(* IEC 61131-3 sources: POMIRTS_lab3/AS/Library_2/ArEthBond, 3 files *)

(* ---- ArEthBond.typ ---- *)
 TYPE
	ArEthBondStateType : STRUCT											(*status data of a bond*)
		ActiveDevice 						: STRING[128];				(*name of the currently active device*)
		PrimaryLinkStatus 					: UDINT;					(*link status of the primary device*)
		SecondaryLinkStatus 				: UDINT;					(*link status of the secondary device*)
		NumberArpReachedTargets 			: UDINT;					(*number of currently reached ARP targets*)
	END_STRUCT;

	ArEthBondStatisticsType : STRUCT									(*statistical data of a bond*)
		SwitchCount 						: UDINT; 					(*number of occurred switches*)
		PrimaryLinkErrorCount 				: UDINT;					(*number of link errors of the primary device*)
		SecondaryLinkErrorCount 			: UDINT;					(*number of link errors of the secondary device*)
		PrimaryArpErrorCount 				: UDINT;					(*number of ARP errors of the primary device*)
		SecondaryArpErrorCount 				: UDINT;					(*number of ARP errors of the secondary device*)
		LastErrorUtcTimeStampSeconds 		: UDINT;					(*seconds part of the last error time stamp*)
		LastErrorUtcTimeStampNanoSeconds 	: UDINT;					(*nano seconds part of the last error time stamp*)
	END_STRUCT;

	ArEthBondConfigurationType : STRUCT
		ArpMonitorPeriodMs 					: UDINT; 					(*period of the ARP monitoring in ms*)
		NumberArpConfiguredTargets 			: UDINT; 					(*number of configured ARP targets*)
	END_STRUCT;

	ArEthBondInternalType : STRUCT
		FBStateCtx							: ArFBStateInternalType; 	(*internal status*)
	END_STRUCT;
END_TYPE

(* ---- ArEthBond.var ---- *)
 VAR CONSTANT
	arETHBOND_ERR_INVALID_NAME 	: DINT := -1070585906;	(*invalid bond name as input parameter*)
END_VAR

(* ---- ArEthBond.fun ---- *)
{REDUND_CONTEXT} {REDUND_UNREPLICABLE} FUNCTION_BLOCK ArEthBondGetData 					 		(*reads data from a bond*)
	VAR_INPUT
		Execute				: BOOL;							(*execute the FB*)
		Name				: STRING[128];					(*name of the bond*)
	END_VAR

	VAR_OUTPUT
		Done	 			: BOOL;							(*execution of the FB finished*)
		Error				: BOOL;							(*execution of the FB failed*)
		ErrorID				: DINT;  						(*error number if execution of the FB has failed*)
		Configuration		: ArEthBondConfigurationType;	(*configuration data of the bond*)
		State				: ArEthBondStateType;			(*status data of the bond*)
		Statistics			: ArEthBondStatisticsType;		(*statistical data of the bond*)
	END_VAR

	VAR
        Internal			: ArEthBondInternalType; 		(*internal variable*)
	END_VAR
END_FUNCTION_BLOCK
